PROGRAM MAIN
VAR
	execute : BOOL;
	stop : BOOL;
	manualStep : BOOL := TRUE;
	manualSuction : BOOL;
	
	moduleWB : WoodBunkEx;
	//moduleCIP : ChipboardEx;
	exec1, exec2 : BOOL;
END_VAR
VAR
	test : BOOL;
END_VAR

SetupHardware();
CallHardwareModules(); //start program with hardware call

moduleWB(
	execute:= exec1, 
	stop:= stop, 
	manualStep:= manualStep, 
	manualSuction:= manualSuction,
 
	robotLeft:= robot1, 
	robotRight:= robot2, 
	toolStorageLeft:= toolStorageA21Left, 
	toolStorageRight:= toolStorageA21Right, 
	stagingTableLeft:= stagingTableLeft, 
	stagingTableRight:= stagingTableRight, 
	magazineLeft:= magazineA21Left, 
	magazineRight:= magazineA21Right, 
	strapper:= strapperA21, 
	horizontalDriveLeft:= horizontalDriveA21Left, 
	horizontalDriveRight:= horizontalDriveA21Right, 
	verticalDriveLeft:= verticalDriveA21Left, 
	verticalDriveRight:= verticalDriveA21Right, 
	pistonBottom:= pistonA21Bottom, 
	topSuction:= suctionA21Top, 
	leftSuction:= suctionA21Left, 
	rightSuction:= suctionA21Right, 
	bottomSuction:= suctionA21Bottom, 
	
	generalError=> test, 
	failLeft=> test, 
	failRight=> test);
(*
moduleCIP(
	execute:= exec2, 
	stop:= stop, 
	manualStep:= manualStep, 
	manualSuction:= manualSuction,
	
	robotLeft:= robot1, 
	robotRight:= robot2, 
	toolStorageLeft:= toolStorageA21Left, 
	toolStorageRight:= toolStorageA21Right, 
	skidLeft:= skidA21Left, 
	skidRight:= skidA21Right, 
	generalError=> test, 
	failLeft=> test, 
	failRight=> test);
*)
CallHardwareModules(); //end program with hardware call

END_PROGRAM

(* stored: Version 1.1.0.1, ProductVersion 3.1.4024.11
   POU MAIN: Id {9caf58b7-eccf-4a65-a3e3-2c8d81beb312}, SpecialFunc None *)
